(* IEC 61131-3 sources: SIMERLIFT/logiwork_simerlift_80v/logiwork_simerlift_80v/HEMAbattery/src_FBD/BCU, 8 files *)

(* ---- ampMaxTemp.iecst ---- *)
FUNCTION_BLOCK ampMultTemp {
    width := 200;
  }

VAR_INPUT
temp:REAL;
END_VAR

VAR_OUTPUT
mult : REAL;
END_VAR

VAR
rstTimer:TON;
timeout:BOOL;
lastMult:REAL;
instantMult:REAL;
END_VAR

IF temp<-20 THEN
	mult:=0;
	instantMult:=0;
ELSIF temp<-15  THEN
	instantMult:=0.1;
ELSIF temp<-10  THEN
	instantMult:=0.15;
ELSIF temp<-5  THEN
	instantMult:=0.2;
ELSIF temp<0  THEN
	instantMult:=0.4;
ELSIF temp<5  THEN
	instantMult:=0.5;
ELSIF temp<10  THEN
	instantMult:=0.7;
ELSIF temp<50  THEN
	instantMult:=1;
ELSIF temp<55  THEN
	instantMult:=0.4;
ELSIF temp<56  THEN
	instantMult:=0.2;
ELSE
	mult:=0;
	instantMult:=0;
END_IF;

rstTimer(IN:=instantMult=lastMult, PT:=T#10s, Q=>timeout);

lastMult:=instantMult;

IF timeout THEN
	mult:=instantMult;
END_IF;

END_FUNCTION_BLOCK

(* ---- ampMultVoltChar.iecst ---- *)
FUNCTION_BLOCK  ampMultVoltChar  {
    width := 200;
  }

VAR_INPUT
    chargeOn:BOOL;
    maxCell:UDINT;
END_VAR

VAR_OUTPUT
	mult:REAL;
END_VAR

VAR
state:USINT;

END_VAR

 IF NOT chargeOn THEN
    state:=0;
 END_IF;

 CASE state OF
	0:
	mult:=1;
	IF maxCell>3350 THEN
		state:=state+1;
	END_IF;

	1:
	mult:=0.7;
	IF maxCell>3400 THEN
		state:=state+1;
	END_IF;

	2:
	mult:=0.6;
	IF maxCell>3450 THEN
		state:=state+1;
	END_IF;

	3:
	mult:=0.5;
	IF maxCell>3500 THEN
		state:=state+1;
	END_IF;

	4:
	mult:=0.35;
	IF maxCell>3550 THEN
		state:=state+1;
	END_IF;

	5:
	mult:=0.3;
	IF maxCell>3600 THEN
		state:=state+1;
	END_IF;

	6:
	mult:=0.2;
	IF maxCell>3650 THEN
		state:=state+1;

	END_IF;

 	7:
	mult:=0;

END_CASE;

 END_FUNCTION_BLOCK

(* ---- ampMultVoltDisc.iecst ---- *)
FUNCTION_BLOCK  ampMultVoltDisc  {
    width := 200;
  }

VAR_INPUT
    discOn:BOOL;
    minCell:UDINT;
END_VAR

VAR_OUTPUT
	mult:REAL;
END_VAR

VAR
state:USINT;

END_VAR

 IF NOT discOn THEN
    state:=0;
 END_IF;

 CASE state OF
	0:
	mult:=1;
	IF minCell<3150 THEN
		state:=state+1;
	END_IF;

	1:
	mult:=0.7;
	IF minCell<3120 THEN
		state:=state+1;
	END_IF;

	2:
	mult:=0.6;
	IF minCell<3100 THEN
		state:=state+1;
	END_IF;

	3:
	mult:=0.5;
	IF minCell<3050 THEN
		state:=state+1;
	END_IF;

	4:
	mult:=0.35;
	IF minCell<3020 THEN
		state:=state+1;
	END_IF;

	5:
	mult:=0.25;
	IF minCell<3000 THEN
		state:=state+1;
	END_IF;

	6:
	mult:=0.2;
	IF minCell<2400 THEN
		state:=state+1;

	END_IF;

 	7:
	mult:=0;

END_CASE;

 END_FUNCTION_BLOCK

(* ---- bessState.iecst ---- *)
FUNCTION_BLOCK  bessState  {
    width := 400;
    bgColor := "mediumseagreen";
  }

VAR_INPUT
	IGNITION : BOOL;
	chargerON:BOOL;
	prechargeOk:BOOL;
	dischargeComplete:BOOL;
	chargeComplete:BOOL;
	shutdownComplete:BOOL;
	contactFbk:BOOL;
	currentAmp:REAL;
	OVfault:BOOL;
    UVfault:BOOL;
	fault:BOOL;
END_VAR

VAR_OUTPUT
	STATE : BATTSTATE;
	prechargeOn:BOOL;
	contact:BOOL;
	contactNeg:BOOL;
END_VAR

VAR
currentCharging:BOOL;
currentDischarging:BOOL;

CURRENTTIMERcharging:TON;
CURRENTTIMERdischarging:TON;

chargeVoltTimer:Tbuffer;
dischargeVoltTimer:Tbuffer;

BATTERYSTATE:BATTSTATE:=BATTSTATE#STANDBY;
PREVSTATE:BATTSTATE:=BATTSTATE#STANDBY;

BATTIMER:TON;
BATSTATEINTERVAL:TIME:=T#10s;
BATSTATETIMEOUT:BOOL;
BATSTATEELAPSEDTIME:TIME;
STANDBYINTERVAL:TIME:=T#2s;
END_VAR

CURRENTTIMERcharging(IN:=currentAmp<-0.5, PT:=T#500ms, Q=>currentCharging);
CURRENTTIMERdischarging(IN:=currentAmp>0.5, PT:=T#500ms, Q=>currentDischarging);
BATTIMER(IN:=BATTERYSTATE=PREVSTATE, PT:=BATSTATEINTERVAL, Q=>BATSTATETIMEOUT, ET=>BATSTATEELAPSEDTIME);

PREVSTATE:=BATTERYSTATE;

CASE BATTERYSTATE OF

	BATTSTATE#STANDBY:  // standby
		STATE:=BATTSTATE#STANDBY;
		BATSTATEINTERVAL:=T#12s;

		prechargeOn:=0;
		contact:=0;
		contactNeg:=0;

		// at the first time wait 2 sec
		IF BATSTATEELAPSEDTIME>STANDBYINTERVAL THEN
		    // then wait 100ms in next sessions
			STANDBYINTERVAL:=T#500ms;
			IF fault THEN
				BATTERYSTATE:=BATTSTATE#FAULT;
			ELSIF IGNITION THEN
				IF chargerON THEN
					IF OVfault OR chargeComplete THEN
						BATTERYSTATE:=BATTSTATE#CHARGECOMPLETE;
					ELSE
						BATTERYSTATE:=BATTSTATE#PRECHARGE;
					END_IF;
				ELSE
					BATTERYSTATE:=BATTSTATE#PRECHARGE;
				END_IF;
			END_IF;

		END_IF;

	BATTSTATE#PRECHARGE:  //discharge
		STATE:=BATTSTATE#PRECHARGE;
		BATSTATEINTERVAL:=T#5s;

		contactNeg:=1;

		IF BATSTATEELAPSEDTIME>T#50ms THEN
			prechargeOn:=1;
		ELSE
			prechargeOn:=0;
		END_IF;

		IF prechargeOk THEN
			contact:=1;
		ELSE
			contact:=0;
		END_IF;

		IF fault OR  NOT IGNITION  THEN
			BATTERYSTATE:=BATTSTATE#SHUTDOWN;
		ELSIF BATSTATETIMEOUT THEN
			BATTERYSTATE:=BATTSTATE#FAULT;
		ELSIF prechargeOk AND contactFbk THEN
			IF chargerON THEN
				IF OVfault OR chargeComplete THEN
					BATTERYSTATE:=BATTSTATE#CHARGECOMPLETE;
				ELSE
					BATTERYSTATE:=BATTSTATE#CHARGE;
				END_IF;
			ELSE
				BATTERYSTATE:=BATTSTATE#DISCHARGE;
			END_IF;
		END_IF;

	BATTSTATE#DISCHARGE:  //discharge
		STATE:=BATTSTATE#DISCHARGE;
		BATSTATEINTERVAL:=T#120s;

		prechargeOn:=0;
		contact:=1;
		contactNeg:=1;

		IF fault OR NOT IGNITION THEN
			BATTERYSTATE:=BATTSTATE#SHUTDOWN;
		ELSIF chargerON THEN
			IF OVfault OR chargeComplete THEN
				BATTERYSTATE:=BATTSTATE#CHARGECOMPLETE;
			ELSE
				BATTERYSTATE:=BATTSTATE#CHARGE;
			END_IF;
		ELSIF BATSTATEELAPSEDTIME>T#10s THEN
			IF currentDischarging THEN
				IF UVfault OR dischargeComplete THEN
					BATTERYSTATE:=BATTSTATE#DISCHARGECOMPLETE;
				END_IF;
			ELSIF currentCharging THEN
				IF OVfault THEN
					BATTERYSTATE:=BATTSTATE#CHARGECOMPLETE;
				END_IF;
			END_IF;
		ELSIF (UVfault OR dischargeComplete) AND currentAmp>10THEN
			BATTERYSTATE:=BATTSTATE#DISCHARGECOMPLETE;
		ELSIF (OVfault OR chargeComplete) AND currentAmp<-10 THEN
			BATTERYSTATE:=BATTSTATE#CHARGECOMPLETE;
		END_IF;

	BATTSTATE#CHARGE:  // charge
		STATE:=BATTSTATE#CHARGE;
		BATSTATEINTERVAL:=T#120s;

		prechargeOn:=0;
		contact:=1;
		contactNeg:=1;

		IF fault OR NOT IGNITION THEN
			BATTERYSTATE:=BATTSTATE#SHUTDOWN;
		ELSIF NOT chargerON THEN
			IF UVfault OR  dischargeComplete THEN
				BATTERYSTATE:=BATTSTATE#DISCHARGECOMPLETE;
			ELSE
				BATTERYSTATE:=BATTSTATE#DISCHARGE;
			END_IF;
		ELSIF OVfault OR chargeComplete THEN
			BATTERYSTATE:=BATTSTATE#CHARGECOMPLETE;
		ELSIF  BATSTATEELAPSEDTIME>T#8s THEN
			IF currentDischarging THEN
				IF UVfault THEN
					BATTERYSTATE:=BATTSTATE#DISCHARGECOMPLETE;
				ELSIF dischargeComplete THEN
					BATTERYSTATE:=BATTSTATE#DISCHARGECOMPLETE;
				END_IF;
			END_IF;
		ELSIF (UVfault OR dischargeComplete) AND currentAmp>10THEN
			BATTERYSTATE:=BATTSTATE#DISCHARGECOMPLETE;
		END_IF;

	BATTSTATE#SHUTDOWN:  // shutdown
		STATE:=BATTSTATE#SHUTDOWN;
		BATSTATEINTERVAL:=T#3000ms;
		prechargeOn:=0;
		IF BATSTATEELAPSEDTIME>T#2500ms OR  (shutdownComplete AND (BATSTATEELAPSEDTIME>T#1000ms))  THEN
			contact:=0;
		 	contactNeg:=0;
		 	IF contactFbk=FALSE THEN
				IF fault THEN
					BATTERYSTATE:=BATTSTATE#FAULT;
				ELSIF UVfault THEN
					BATTERYSTATE:=BATTSTATE#DISCHARGECOMPLETE;
				ELSIF OVfault THEN
					BATTERYSTATE:=BATTSTATE#CHARGECOMPLETE;
				ELSIF NOT IGNITION THEN
					BATTERYSTATE:=BATTSTATE#STANDBY;
				END_IF;
			ELSIF BATSTATEELAPSEDTIME>T#2800ms THEN
				BATTERYSTATE:=BATTSTATE#FAULT;
			END_IF;

		END_IF;

	BATTSTATE#FAULT:  //fault
		STATE:=BATTSTATE#FAULT;
		BATSTATEINTERVAL:=T#10s;

		prechargeOn:=0;
		contact:=0;
		contactNeg:=0;

		IF NOT fault AND (NOT IGNITION OR BATSTATETIMEOUT) THEN
			BATTERYSTATE:=BATTSTATE#STANDBY;
		END_IF;

	BATTSTATE#CHARGECOMPLETE:  //charge complete
		STATE:=BATTSTATE#CHARGECOMPLETE;
		BATSTATEINTERVAL:=T#5s;

		prechargeOn:=0;
		contact:=0;
		contactNeg:=0;

		IF fault OR NOT IGNITION THEN
			BATTERYSTATE:=BATTSTATE#SHUTDOWN;
		ELSIF NOT chargerON AND BATSTATETIMEOUT THEN
			IF UVfault THEN
				BATTERYSTATE:=BATTSTATE#DISCHARGECOMPLETE;
			ELSIF dischargeComplete THEN
				BATTERYSTATE:=BATTSTATE#DISCHARGECOMPLETE;
			ELSE
				BATTERYSTATE:=BATTSTATE#PRECHARGE;
			END_IF;
		END_IF;

	BATTSTATE#DISCHARGECOMPLETE:  //charge complete
		STATE:=BATTSTATE#DISCHARGECOMPLETE;
		BATSTATEINTERVAL:=T#5s;

		prechargeOn:=0;
		contact:=0;
		contactNeg:=0;

		IF fault THEN
			BATTERYSTATE:=BATTSTATE#SHUTDOWN;
		ELSIF NOT IGNITION THEN
			BATTERYSTATE:=BATTSTATE#SHUTDOWN;
		ELSIF chargerON AND BATSTATETIMEOUT THEN
			IF OVfault THEN
				BATTERYSTATE:=BATTSTATE#CHARGECOMPLETE;
			ELSIF chargeComplete THEN
				BATTERYSTATE:=BATTSTATE#CHARGECOMPLETE;
			ELSE
				BATTERYSTATE:=BATTSTATE#PRECHARGE;   /// because no current will flow unless contact closed
			END_IF;
		END_IF;

END_CASE;

END_FUNCTION_BLOCK

(* ---- chargeState.iecst ---- *)
FUNCTION_BLOCK  chargeState  {
    width := 400;
  }

VAR_INPUT
    chargeOn:BOOL;
    mainComplete:BOOL;
    dmcc:REAL;
	battAmpr:REAL;
	balAmpr:REAL;
	balDiff:UDINT;
    maxCell:UDINT;
    minCell:UDINT;
END_VAR

VAR_OUTPUT
	complete:BOOL;
	balance:BOOL;
	chargeAmpr:REAL;
	chState:USINT;
END_VAR

VAR

balDiffTol:UDINT;

balanceOK_mid:BOOL;
balanceOK:BOOL;
balanceTIMERhigh:TON;
balanceTIMERlow:TOF;

amperLow_mid:BOOL;
amperLow:BOOL;
amperTIMERhigh:TON;
amperTIMERlow:TOF;

PREVSTATE:USINT:=0;
state:USINT;
chargeTIMER:TON;
chargeInterval:TIME:=T#1s;
chargeSTATETIMEOUT:BOOL;
chargeSTATEELAPSEDTIME:TIME;
END_VAR

chargeTIMER(IN:=state=PREVSTATE, PT:=chargeInterval, Q=>chargeSTATETIMEOUT, ET=>chargeSTATEELAPSEDTIME);
PREVSTATE:=state;

amperTIMERhigh(IN:=ABS(battAmpr)<(balAmpr+3), PT:=T#3s, Q=>amperLow_mid);
amperTIMERlow(IN:=amperLow_mid, PT:=T#3s, Q=>amperLow);

balanceTIMERhigh(IN:= (maxCell-minCell)<balDiffTol, PT:=T#5s, Q=>balanceOK_mid);  //20
balanceTIMERlow(IN:=balanceOK_mid, PT:=T#5s, Q=>balanceOK);  //20

 IF NOT chargeOn THEN
    state:=0;
END_IF;

CASE state OF

	0: //stb
	chargeInterval:=T#5m;
	complete:=mainComplete;
	balance:=0;
	chargeAmpr:=dmcc;

	IF chargeOn AND NOT complete THEN
		state:=1;
		complete:=0;
	END_IF;

	1: //charge on
	chargeInterval:=T#5m;  //5m
	complete:=0;
	balance:=0;
	chargeAmpr:=dmcc;
	IF mainComplete THEN
		state:=2;  // go to rest before balance decision
	END_IF;

	2:  //rest
	chargeInterval:=T#10s;  //2m
	complete:=0;
	balance:=0;
	chargeAmpr:=balAmpr;
	balDiffTol:=balDiff;

	IF chargeSTATETIMEOUT THEN
		IF balanceOK THEN
			state:=4;
		ELSE
			state:=3;
		END_IF;
	ELSIF chargeSTATEELAPSEDTIME>T#30s THEN
		IF NOT amperLow THEN
			state:=4;
		END_IF;
	END_IF;

	3:  //balance
	chargeInterval:=T#1m;  //30m
	complete:=0;
	balance:=1;
	chargeAmpr:=balAmpr;
	balDiffTol:=10;

	IF chargeSTATETIMEOUT OR NOT amperLow THEN
		state:=4;
	ELSIF chargeSTATEELAPSEDTIME>T#10m THEN   //10m
		IF balanceOK THEN
			state:=4;
		END_IF;
	END_IF;

	4: //charge state complete
	chargeInterval:=T#1m;   //1m
	complete:=1;
	balance:=0;
	chargeAmpr:=0;

END_CASE;

chState:=state;

END_FUNCTION_BLOCK

(* ---- Current.iecfbd ---- *)
FUNCTION_BLOCK Current
  {
    Current {index := 0};
    Discharge_Current {index := 0};
    Charge_Current {index := 1};
    width := 300;
    height := 38;
  }

  VAR_INPUT
    Current : REAL := 0;
  END_VAR
  VAR_OUTPUT
    Charge_Current : UINT := 0;
    Discharge_Current : UINT := 0;
  END_VAR

  (*

    // Network 1:
    DIV(IN1 := Current, IN2 := 1000, DIV => @C(2).DIV);
    GE(IN1 := @C(2).DIV, IN2 := 0, GE => @C(11).GE);
    SEL_REAL(G := @C(11).GE, IN0 := 0, IN1 := @C(2).DIV, SEL_REAL => @C(19).SEL_REAL);
    TO_UINT(IN := @C(19).SEL_REAL, TO_UINT => Discharge_Current);
    LT(IN1 := @C(2).DIV, IN2 := 0, LT => @C(15).LT);
    MUL(IN1 := @C(2).DIV, IN2 := -1, MUL => @C(34).MUL);
    SEL_REAL(G := @C(15).LT, IN0 := 0, IN1 := @C(34).MUL, SEL_REAL => @C(27).SEL_REAL);
    TO_UINT(IN := @C(27).SEL_REAL, TO_UINT => Charge_Current);

  *)

  @VF(1) : @E(Current), @R(20.0, 20.0, 220.0, 19.0);
  @VF(4) : @E(Charge_Current), @R(1100.0, 80.0, 220.0, 19.0);
  @VF(5) : @E(Discharge_Current), @R(1100.0, 20.0, 220.0, 19.0);
  @C(11) : @F(GE), @R(550.0, 20.0, 40.0, 38.0), REAL, @I(@N(IN1), @L(9.5)), @I(@N(IN2), @L(29.5)), @O(@N(GE), @R(9.5));
  @VF(13) : @E(0), @R(360.0, 40.0, 110.0, 19.0), REAL;
  @C(15) : @F(LT), @R(550.0, 80.0, 40.0, 38.0), REAL, @I(@N(IN1), @L(9.5)), @I(@N(IN2), @L(29.5)), @O(@N(LT), @R(9.5));
  @VF(17) : @E(0), @R(360.0, 100.0, 110.0, 19.0), REAL;
  @C(19) : @F(SEL_REAL), @R(780.0, 20.0, 120.0, 58.0), @I(@N(G), @L(9.5)), @I(@N(IN0), @L(29.5)), @I(@N(IN1), @L(49.5)), @O(@N(SEL_REAL), @R(9.5));
  @VF(21) : @E(0), @R(630.0, 40.0, 110.0, 19.0), REAL;
  @C(24) : @F(TO_UINT), @R(940.0, 20.0, 120.0, 18.0), REAL, @I(@N(IN), @L(9.5)), @O(@N(TO_UINT), @R(9.5));
  @C(27) : @F(SEL_REAL), @R(780.0, 80.0, 120.0, 58.0), @I(@N(G), @L(9.5)), @I(@N(IN0), @L(29.5)), @I(@N(IN1), @L(49.5)), @O(@N(SEL_REAL), @R(9.5));
  @VF(28) : @E(0), @R(630.0, 100.0, 110.0, 19.0), REAL;
  @C(31) : @F(TO_UINT), @R(940.0, 80.0, 120.0, 18.0), REAL, @I(@N(IN), @L(9.5)), @O(@N(TO_UINT), @R(9.5));
  @C(34) : @F(MUL), @R(550.0, 120.0, 40.0, 38.0), REAL, @I(@N(IN1), @L(9.5)), @I(@N(IN2), @L(29.5)), @O(@N(MUL), @R(9.5));
  @VF(37) : @E(-1), @R(360.0, 140.0, 110.0, 19.0), REAL;
  @C(2) : @F(DIV), @R(280.0, 20.0, 40.0, 38.0), REAL, @I(@N(IN1), @L(9.5)), @I(@N(IN2), @L(29.5)), @O(@N(DIV), @R(9.5));
  @VF(7) : @E(1000), @R(130.0, 40.0, 110.0, 19.0), REAL;
  @CP(16) : 509.5, 29.5;
  @CP(23) : 509.5, 69.5;
  @CP(35) : 509.5, 89.5;

  @G(6) :
     @L(@CP(16), @C(11).IN1),
     @L(@CP(16), @CP(23)),
     @L(@CP(23), @CP(35)),
     @L(@CP(23), @C(19).IN1),
     @L(@CP(35), @C(15).IN1),
     @L(@CP(35), @C(34).IN1),
     @L(@C(2).DIV, @CP(16))
    ;
  @G(14) :
     @L(@VF(13).o, @C(11).IN2)
    ;
  @G(18) :
     @L(@VF(17).o, @C(15).IN2)
    ;
  @G(20) :
     @L(@C(11).GE, @C(19).G)
    ;
  @G(22) :
     @L(@VF(21).o, @C(19).IN0)
    ;
  @G(25) :
     @L(@C(19).SEL_REAL, @C(24).IN)
    ;
  @G(26) :
     @L(@C(24).TO_UINT, @VF(5).i)
    ;
  @G(29) :
     @L(@VF(28).o, @C(27).IN0)
    ;
  @G(30) :
     @L(@C(15).LT, @C(27).G)
    ;
  @G(32) :
     @L(@C(27).SEL_REAL, @C(31).IN)
    ;
  @G(33) :
     @L(@C(31).TO_UINT, @VF(4).i)
    ;
  @G(36) :
     @L(@C(34).MUL, @C(27).IN1)
    ;
  @G(38) :
     @L(@VF(37).o, @C(34).IN2)
    ;
  @G(3) :
     @L(@VF(1).o, @C(2).IN1)
    ;
  @G(8) :
     @L(@VF(7).o, @C(2).IN2)
    ;
END_FUNCTION_BLOCK

(* ---- essState1.iecst ---- *)
FUNCTION_BLOCK  essState1  {
    fault {index := 12};
    shutdownComplete {index := 11};
    chargeProtect {index := 9};
    dischargeProtect {index := 8};
    contactFbkNeg {loc := "left", index := 6};
    contactFbk {loc := "left", index := 5};
    prechargeOk {loc := "left", index := 4};
    contactNeg {loc := "right", index := 4};
    contact {loc := "right", index := 3};
    prechargeOn {loc := "right", index := 2};
    width := 400;
    bgColor := "mediumseagreen";
    height := 258;
  }

VAR_INPUT
	discharge:BOOL;
	charge:BOOL;
	shutdown:BOOL;

	prechargeOk:BOOL;
	contactFbk:BOOL;
	contactFbkNeg:BOOL;

	dischargeProtect:BOOL;
	chargeProtect:BOOL;

	shutdownComplete:BOOL;
	fault:BOOL;
END_VAR

VAR_OUTPUT
	STATE : BATTSTATE;

	prechargeOn:BOOL;
	contact:BOOL;
	contactNeg:BOOL;
END_VAR

VAR

BATTERYSTATE:BATTSTATE:=BATTSTATE#STANDBY;
PREVSTATE:BATTSTATE:=BATTSTATE#STANDBY;

BATTIMER:TON;
BATSTATEINTERVAL:TIME:=T#10s;
BATSTATETIMEOUT:BOOL;
BATSTATEELAPSEDTIME:TIME;
STANDBYINTERVAL:TIME:=T#2s;
END_VAR

BATTIMER(IN:=BATTERYSTATE=PREVSTATE, PT:=BATSTATEINTERVAL, Q=>BATSTATETIMEOUT, ET=>BATSTATEELAPSEDTIME);

PREVSTATE:=BATTERYSTATE;

CASE BATTERYSTATE OF

	BATTSTATE#STANDBY:  // standby
		STATE:=BATTSTATE#STANDBY;
		BATSTATEINTERVAL:=T#12s;

		contact:=0;
		contactNeg:=0;
		prechargeOn:=0;

        IF BATSTATEELAPSEDTIME>STANDBYINTERVAL THEN
        	STANDBYINTERVAL:=T#500ms;
        	IF fault THEN
				BATTERYSTATE:=BATTSTATE#FAULT;
			ELSIF shutdown THEN
				BATTERYSTATE:=BATTSTATE#SHUTDOWN;
			ELSIF discharge OR (charge AND NOT chargeProtect) THEN
				BATTERYSTATE:=BATTSTATE#PRECHARGE;
			END_IF;
        END_IF;

	BATTSTATE#PRECHARGE:  //discharge
		STATE:=BATTSTATE#PRECHARGE;
		BATSTATEINTERVAL:=T#5s;

		contactNeg:=1;

		IF BATSTATEELAPSEDTIME>T#50ms AND contactFbkNeg THEN
			prechargeOn:=1;
		END_IF;

		IF prechargeOk THEN
			contact:=1;
		END_IF;

		IF fault OR NOT(discharge OR charge) OR shutdown OR BATSTATETIMEOUT THEN
			BATTERYSTATE:=BATTSTATE#SHUTDOWN;
		ELSIF prechargeOk AND contactFbk AND contactFbkNeg THEN
			IF charge THEN
				BATTERYSTATE:=BATTSTATE#CHARGE;
			ELSE
				BATTERYSTATE:=BATTSTATE#DISCHARGE;
			END_IF;
		END_IF;

	BATTSTATE#DISCHARGE:  //discharge
		STATE:=BATTSTATE#DISCHARGE;
		BATSTATEINTERVAL:=T#120s;

		prechargeOn:=0;
		contact:=1;
		contactNeg:=1;

		IF fault OR shutdown OR NOT contactFbk OR NOT contactFbkNeg THEN
			BATTERYSTATE:=BATTSTATE#SHUTDOWN;
		ELSIF NOT discharge THEN
			IF charge AND NOT chargeProtect THEN
				BATTERYSTATE:=BATTSTATE#CHARGE;
			ELSE
				BATTERYSTATE:=BATTSTATE#SHUTDOWN;
			END_IF;
		END_IF;

	BATTSTATE#CHARGE:  // charge
		STATE:=BATTSTATE#CHARGE;
		BATSTATEINTERVAL:=T#120s;

		prechargeOn:=0;
		contact:=1;
		contactNeg:=1;

		IF fault OR shutdown OR NOT contactFbk OR NOT contactFbkNeg THEN
			BATTERYSTATE:=BATTSTATE#SHUTDOWN;
		ELSIF NOT charge THEN
			IF discharge THEN
				BATTERYSTATE:=BATTSTATE#DISCHARGE;
			ELSE
				BATTERYSTATE:=BATTSTATE#SHUTDOWN;
			END_IF;
		END_IF;

	BATTSTATE#SHUTDOWN:  // shutdown
		STATE:=BATTSTATE#SHUTDOWN;
		BATSTATEINTERVAL:=T#5000ms;

		prechargeOn:=0;

		IF shutdown OR BATSTATEELAPSEDTIME>T#2000ms OR (shutdownComplete AND (BATSTATEELAPSEDTIME>T#500ms))  THEN
			contact:=0;
			contactNeg:=0;
			IF fault THEN
				BATTERYSTATE:=BATTSTATE#FAULT;
			ELSIF shutdown THEN
				BATTERYSTATE:=BATTSTATE#SHUTDOWN;
			ELSIF NOT contactFbk AND NOT contactFbkNeg THEN
				IF dischargeProtect THEN
					BATTERYSTATE:=BATTSTATE#DISCHARGECOMPLETE;
				ELSIF chargeProtect THEN
					BATTERYSTATE:=BATTSTATE#CHARGECOMPLETE;
				ELSIF BATSTATETIMEOUT OR charge OR discharge THEN
					BATTERYSTATE:=BATTSTATE#STANDBY;
				END_IF;
			END_IF;
		END_IF;

	BATTSTATE#FAULT:  //fault
		STATE:=BATTSTATE#FAULT;
		BATSTATEINTERVAL:=T#10s;

		contact:=0;
		contactNeg:=0;
		prechargeOn:=0;

		IF NOT fault AND BATSTATETIMEOUT THEN
			BATTERYSTATE:=BATTSTATE#SHUTDOWN;
		END_IF;

	BATTSTATE#CHARGECOMPLETE:
		STATE:=BATTSTATE#CHARGECOMPLETE;
		BATSTATEINTERVAL:=T#5s;

		prechargeOn:=0;
		contact:=0;
		contactNeg:=0;

		IF fault THEN
			BATTERYSTATE:=BATTSTATE#FAULT;
		ELSIF shutdown THEN
			BATTERYSTATE:=BATTSTATE#SHUTDOWN;
		ELSIF BATSTATETIMEOUT AND discharge THEN
			BATTERYSTATE:=BATTSTATE#STANDBY;
		END_IF;

	BATTSTATE#DISCHARGECOMPLETE:
		STATE:=BATTSTATE#DISCHARGECOMPLETE;
		BATSTATEINTERVAL:=T#5s;

		prechargeOn:=0;
		contact:=0;
		contactNeg:=0;

		IF fault THEN
			BATTERYSTATE:=BATTSTATE#FAULT;
		ELSIF shutdown THEN
			BATTERYSTATE:=BATTSTATE#SHUTDOWN;
		ELSIF BATSTATETIMEOUT AND charge THEN
			BATTERYSTATE:=BATTSTATE#STANDBY;
		END_IF;

END_CASE;

END_FUNCTION_BLOCK

(* ---- GUI.iecfbd ---- *)
FUNCTION_BLOCK GUI
  {
    SoC {index := 0};
    SoH {index := 1};
    Voltage {index := 2};
    Current {index := 3};
    Temp {index := 4};
    Humidity {index := 5};
    Fault {index := 6};
    width := 200;
    height := 138;
  }

  VAR
    TP1 : TP;
    BAMTX2 : BAMTX;
    BATTSTACKinfo1 : BATTSTACKinfo;
    CANRECV5 : CANRECV;
    tauxCells : ARRAY[0..15] OF USINT := [0,0,0,1,1,1,2,2,2,3,3,3,4,4,4,4];
    guiReqCount : UDINT;
  END_VAR
  VAR_INPUT
    Voltage : REAL := 0;
    Current : REAL := 0;
    Temp : REAL := 0;
    Humidity : REAL := 0;
    Fault : UDINT := 0;
    SoC : USINT := 0;
    SoH : USINT := 0;
    Cycle : UINT;
    State : USINT;
    ID : USINT;
    CH : TMS570_CAN;
  END_VAR

  (*

    // Network 1:
    CANRECV5(CH := CH, ID := 16#18EA1EA4, FMT := CAN_FORMAT#EXTENDED, PER := T#1s, ENB := 1);
    RBIT(start := 0, len := 16, INbit := CANRECV5.DATA, OUTbit => @C(31).OUTbit);
    TO_UINT(IN := @C(31).OUTbit, TO_UINT => @C(2560).TO_UINT);
    FROM_BIG_ENDIAN(IN := @C(2560).TO_UINT, FROM_BIG_ENDIAN => @C(774).FROM_BIG_ENDIAN);
    RBIT(start := 8, len := 8, INbit := CANRECV5.DATA, OUTbit => @C(35).OUTbit);
    TO_USINT(IN := @C(35).OUTbit, TO_USINT => @C(2558).TO_USINT);
    RBIT(start := 0, len := 4, INbit := CANRECV5.DATA, OUTbit => @C(36).OUTbit);
    TO_USINT(IN := @C(36).OUTbit, TO_USINT => @C(2559).TO_USINT);
    DIV(IN1 := Voltage, IN2 := 1000, DIV => @C(988).DIV);
    DIV(IN1 := Current, IN2 := 1000, DIV => @C(12).DIV);
    TO_SINT(IN := Temp, TO_SINT => @C(799).TO_SINT);
    TO_USINT(IN := Humidity, TO_USINT => @C(820).TO_USINT);
    RBIT(start := 4, len := 4, INbit := CANRECV5.DATA, OUTbit => @C(29).OUTbit);
    TO_USINT(IN := @C(29).OUTbit, TO_USINT => @C(27).TO_USINT);
    EQ(IN1 := @C(27).TO_USINT, IN2 := ID, EQ => @C(789).EQ);
    NE(IN1 := guiReqCount, IN2 := CANRECV5.CRX, NE => @C(2565).NE);
    SEL(G := @C(2565).NE, IN0 := guiReqCount, IN1 := CANRECV5.CRX, SEL => guiReqCount);
    AND(IN1 := @C(2565).NE, IN2 := @C(789).EQ, AND => @C(779).AND);
    BATTSTACKinfo1(INFO := @C(2558).TO_USINT, BRD := @C(2559).TO_USINT, volt := @C(988).DIV, amp := @C(12).DIV, Cycle := Cycle, State := State, SOC := SoC, SOH := SoH, temp := @C(799).TO_SINT, hum := @C(820).TO_USINT, fault := Fault, NTCBETA := 3950, NTCNOMT_KLV := 298.15, NTCNOMR_OHM := 10000.0, T_CELLS := tAuxCells, R := @C(779).AND);
    BAMTX2(CH := CH, TPCM := 16#18FFABCD, TPDT := 16#18FFABCE, PGN := @C(774).FROM_BIG_ENDIAN, FRMPER := T#50ms, DATA := BATTSTACKinfo1.DATA, LEN := BATTSTACKinfo1.LEN, R := BATTSTACKinfo1.R_OUT);
    TP1(IN := BAMTX2.R_END, PT := T#100ms);

  *)

  @C(771) : @FB(TP1), @R(1640.0, 100.0, 100.0, 38.0), @I(@N(IN), @L(9.5)), @I(@N(PT), @L(29.5)), @O(@N(Q), @R(9.5)), @O(@N(ET), @R(29.5));
  @C(2566) : @FB(BAMTX2), @R(1290.0, 60.0, 220.0, 158.0), @I(@N(CH), @L(9.5)), @I(@N(TPCM), @L(29.5)), @I(@N(TPDT), @L(49.5)), @I(@N(PGN), @L(69.5)), @I(@N(FRMPER), @L(89.5)), @I(@N(DATA), @L(109.5)), @I(@N(LEN), @L(129.5)), @I(@N(R), @L(149.5)), @O(@N(CTX), @R(9.5)), @O(@N(RC), @R(29.5)), @O(@N(R_END), @R(49.5));
  @C(774) : @F(FROM_BIG_ENDIAN), @R(1110.0, 120.0, 160.0, 18.0), UINT, @I(@N(IN), @L(9.5)), @O(@N(FROM_BIG_ENDIAN), @R(9.5));
  @C(779) : @F(AND), @R(910.0, 460.0, 40.0, 38.0), BOOL, @I(@N(IN1), @L(9.5)), @I(@N(IN2), @L(29.5)), @O(@N(AND), @R(9.5));
  @C(789) : @F(EQ), @R(850.0, 480.0, 40.0, 38.0), USINT, @I(@N(IN1), @L(9.5)), @I(@N(IN2), @L(29.5)), @O(@N(EQ), @R(9.5));
  @C(799) : @F(TO_SINT), @R(840.0, 320.0, 110.0, 18.0), REAL, @I(@N(IN), @L(9.5)), @O(@N(TO_SINT), @R(9.5));
  @C(820) : @F(TO_USINT), @R(840.0, 340.0, 110.0, 18.0), REAL, @I(@N(IN), @L(9.5)), @O(@N(TO_USINT), @R(9.5));
  @C(2564) : @F(SEL), @R(690.0, 40.0, 120.0, 58.0), UDINT, @I(@N(G), @L(9.5)), @I(@N(IN0), @L(29.5)), @I(@N(IN1), @L(49.5)), @O(@N(SEL), @R(9.5));
  @C(2558) : @F(TO_USINT), @R(840.0, 160.0, 110.0, 18.0), LWORD, @I(@N(IN), @L(9.5)), @O(@N(TO_USINT), @R(9.5));
  @C(2559) : @F(TO_USINT), @R(840.0, 180.0, 110.0, 18.0), LWORD, @I(@N(IN), @L(9.5)), @O(@N(TO_USINT), @R(9.5));
  @C(2560) : @F(TO_UINT), @R(840.0, 120.0, 110.0, 18.0), LWORD, @I(@N(IN), @L(9.5)), @O(@N(TO_UINT), @R(9.5));
  @C(2565) : @F(NE), @R(410.0, 40.0, 40.0, 38.0), UDINT, @I(@N(IN1), @L(9.5)), @I(@N(IN2), @L(29.5)), @O(@N(NE), @R(9.5));
  @C(2567) : @FB(CANRECV5), @R(210.0, 120.0, 160.0, 98.0), @I(@N(CH), @L(9.5)), @I(@N(ID), @L(29.5)), @I(@N(FMT), @L(49.5)), @I(@N(PER), @L(69.5)), @I(@N(ENB), @L(89.5)), @O(@N(CRX), @R(9.5)), @O(@N(DATA), @R(29.5)), @O(@N(DLC), @R(49.5)), @O(@N(MPER), @R(69.5)), @O(@N(RC), @R(89.5));
  @VF(791) : @E(T#100ms), @R(1530.0, 120.0, 90.0, 19.0);
  @VF(2577) : @E(T#50ms), @R(1160.0, 140.0, 110.0, 19.0);
  @VF(2580) : @E(16#18FFABCE), @R(1050.0, 100.0, 220.0, 19.0), UDINT;
  @VF(2586) : @E(16#18FFABCD), @R(1050.0, 80.0, 220.0, 19.0), UDINT;
  @VF(2572) : @E(tAuxCells), @R(840.0, 440.0, 110.0, 19.0);
  @VF(2573) : @E(298.15), @R(840.0, 400.0, 110.0, 19.0), REAL;
  @VF(2575) : @E(10000.0), @R(840.0, 420.0, 110.0, 19.0), REAL;
  @VF(793) : @E(3950), @R(840.0, 380.0, 110.0, 19.0), REAL;
  @VF(837) : @E(guiReqCount), @R(480.0, 60.0, 110.0, 19.0);
  @VF(2581) : @E(0), @R(410.0, 100.0, 40.0, 19.0), INT;
  @VF(2583) : @E(8), @R(410.0, 180.0, 40.0, 19.0), INT;
  @VF(2582) : @E(8), @R(410.0, 160.0, 40.0, 19.0), INT;
  @VF(2578) : @E(16), @R(410.0, 120.0, 40.0, 19.0), INT;
  @VF(2585) : @E(4), @R(410.0, 240.0, 40.0, 19.0), INT;
  @VF(2584) : @E(0), @R(410.0, 220.0, 40.0, 19.0), INT;
  @VF(801) : @E(4), @R(410.0, 480.0, 40.0, 19.0), INT;
  @VF(802) : @E(4), @R(410.0, 500.0, 40.0, 19.0), INT;
  @VF(798) : @E(guiReqCount), @R(280.0, 40.0, 110.0, 19.0);
  @VF(2592) : @E(1), @R(80.0, 200.0, 110.0, 19.0), BOOL;
  @VF(2591) : @E(T#1s), @R(80.0, 180.0, 110.0, 19.0);
  @VF(2593) : @E(CAN_FORMAT#EXTENDED), @R(20.0, 160.0, 170.0, 19.0);
  @VF(2589) : @E(16#18EA1EA4), @R(20.0, 140.0, 170.0, 19.0), UDINT;
  @VF(1) : @E(Fault), @R(840.0, 360.0, 110.0, 19.0);
  @VF(2) : @E(Humidity), @R(730.0, 340.0, 90.0, 19.0);
  @VF(3) : @E(Temp), @R(730.0, 320.0, 90.0, 19.0);
  @VF(4) : @E(Current), @R(20.0, 320.0, 220.0, 19.0);
  @VF(5) : @E(Voltage), @R(20.0, 280.0, 220.0, 19.0);
  @VF(6) : @E(SoC), @R(840.0, 280.0, 110.0, 19.0);
  @VF(7) : @E(SoH), @R(840.0, 300.0, 110.0, 19.0);
  @C(988) : @F(DIV), @R(280.0, 280.0, 40.0, 38.0), REAL, @I(@N(IN1), @L(9.5)), @I(@N(IN2), @L(29.5)), @O(@N(DIV), @R(9.5));
  @VF(981) : @E(1000), @R(130.0, 300.0, 110.0, 19.0), REAL;
  @C(12) : @F(DIV), @R(280.0, 320.0, 40.0, 38.0), REAL, @I(@N(IN1), @L(9.5)), @I(@N(IN2), @L(29.5)), @O(@N(DIV), @R(9.5));
  @VF(16) : @E(1000), @R(130.0, 340.0, 110.0, 19.0), REAL;
  @VF(21) : @E(Cycle), @R(840.0, 240.0, 110.0, 19.0);
  @VF(22) : @E(State), @R(840.0, 260.0, 110.0, 19.0);
  @C(773) : @FB(BATTSTACKinfo1), @R(970.0, 160.0, 300.0, 318.0), @I(@N(INFO), @L(9.5)), @I(@N(BRD), @L(29.5)), @I(@N(volt), @L(49.5)), @I(@N(amp), @L(69.5)), @I(@N(Cycle), @L(89.5)), @I(@N(State), @L(109.5)), @I(@N(SOC), @L(129.5)), @I(@N(SOH), @L(149.5)), @I(@N(temp), @L(169.5)), @I(@N(hum), @L(189.5)), @I(@N(fault), @L(209.5)), @I(@N(NTCBETA), @L(229.5)), @I(@N(NTCNOMT_KLV), @L(249.5)), @I(@N(NTCNOMR_OHM), @L(269.5)), @I(@N(T_CELLS), @L(289.5)), @I(@N(R), @L(309.5)), @O(@N(DATA), @R(9.5)), @O(@N(LEN), @R(29.5)), @O(@N(R_OUT), @R(49.5));
  @VF(25) : @E(ID), @R(660.0, 500.0, 140.0, 19.0);
  @C(27) : @F(TO_USINT), @R(670.0, 480.0, 120.0, 18.0), LWORD, @I(@N(IN), @L(9.5)), @O(@N(TO_USINT), @R(9.5));
  @VF(32) : @E(CH), @R(10.0, 10.0, 140.0, 19.0);
  @C(31) : @F(RBIT), @R(470.0, 100.0, 120.0, 58.0), @I(@N(start), @L(9.5)), @I(@N(len), @L(29.5)), @I(@N(INbit), @L(49.5)), @O(@N(OUTbit), @R(9.5));
  @C(35) : @F(RBIT), @R(470.0, 160.0, 120.0, 58.0), @I(@N(start), @L(9.5)), @I(@N(len), @L(29.5)), @I(@N(INbit), @L(49.5)), @O(@N(OUTbit), @R(9.5));
  @C(36) : @F(RBIT), @R(470.0, 220.0, 120.0, 58.0), @I(@N(start), @L(9.5)), @I(@N(len), @L(29.5)), @I(@N(INbit), @L(49.5)), @O(@N(OUTbit), @R(9.5));
  @C(29) : @F(RBIT), @R(470.0, 480.0, 120.0, 58.0), @I(@N(start), @L(9.5)), @I(@N(len), @L(29.5)), @I(@N(INbit), @L(49.5)), @O(@N(OUTbit), @R(9.5));
  @CP(804) : 619.5, 49.5;
  @CP(2595) : 389.5, 149.5;
  @CP(58) : 389.5, 209.5;
  @CP(282) : 389.5, 269.5;
  @CP(333) : 389.5, 89.5;
  @CP(34) : 189.5, 19.5;

  @G(805) :
     @L(@VF(791).o, @C(771).PT)
    ;
  @G(825) :
     @L(@C(2566).R_END, @C(771).IN)
    ;
  @G(2612) :
     @L(@VF(2577).o, @C(2566).FRMPER)
    ;
  @G(2622) :
     @L(@VF(2580).o, @C(2566).TPDT)
    ;
  @G(2629) :
     @L(@VF(2586).o, @C(2566).TPCM)
    ;
  @G(828) :
     @L(@C(774).FROM_BIG_ENDIAN, @C(2566).PGN)
    ;
  @G(823) :
     @L(@C(773).DATA, @C(2566).DATA)
    ;
  @G(821) :
     @L(@C(773).LEN, @C(2566).LEN)
    ;
  @G(817) :
     @L(@C(773).R_OUT, @C(2566).R)
    ;
  @G(807) :
     @L(@C(799).TO_SINT, @C(773).temp)
    ;
  @G(834) :
     @L(@C(820).TO_USINT, @C(773).hum)
    ;
  @G(813) :
     @L(@VF(793).o, @C(773).NTCBETA)
    ;
  @G(814) :
     @L(@VF(2573).o, @C(773).NTCNOMT_KLV)
    ;
  @G(815) :
     @L(@VF(2575).o, @C(773).NTCNOMR_OHM)
    ;
  @G(816) :
     @L(@VF(2572).o, @C(773).T_CELLS)
    ;
  @G(824) :
     @L(@C(779).AND, @C(773).R)
    ;
  @G(819) :
     @L(@C(2559).TO_USINT, @C(773).BRD)
    ;
  @G(822) :
     @L(@C(2558).TO_USINT, @C(773).INFO)
    ;
  @G(829) :
     @L(@C(2560).TO_UINT, @C(774).IN)
    ;
  @G(2628) :
     @L(@C(2565).NE, @CP(804)),
     @L(@CP(804), @C(2564).G),
     @L(@CP(804), @C(779).IN1)
    ;
  @G(838) :
     @L(@VF(837).o, @C(2564).IN0)
    ;
  @G(2618) :
     @L(@C(2567).CRX, @CP(333)),
     @L(@CP(333), @C(2565).IN2),
     @L(@CP(333), @C(2564).IN1)
    ;
  @G(2621) :
     @L(@C(2567).DATA, @CP(2595)),
     @L(@CP(2595), @CP(58)),
     @L(@CP(58), @CP(282)),
     @L(@CP(282), @C(36).INbit),
     @L(@CP(58), @C(35).INbit),
     @L(@CP(2595), @C(31).INbit),
     @L(@CP(282), @C(29).INbit)
    ;
  @G(812) :
     @L(@VF(798).o, @C(2565).IN1)
    ;
  @G(836) :
     @L(@C(2564).SEL, @VF(798).i)
    ;
  @G(2633) :
     @L(@VF(2593).o, @C(2567).FMT)
    ;
  @G(2634) :
     @L(@VF(2589).o, @C(2567).ID)
    ;
  @G(2635) :
     @L(@VF(2591).o, @C(2567).PER)
    ;
  @G(2636) :
     @L(@VF(2592).o, @C(2567).ENB)
    ;
  @G(8) :
     @L(@VF(1).o, @C(773).fault)
    ;
  @G(9) :
     @L(@VF(3).o, @C(799).IN)
    ;
  @G(10) :
     @L(@VF(2).o, @C(820).IN)
    ;
  @G(13) :
     @L(@VF(6).o, @C(773).SOC)
    ;
  @G(14) :
     @L(@VF(7).o, @C(773).SOH)
    ;
  @G(15) :
     @L(@VF(981).o, @C(988).IN2)
    ;
  @G(11) :
     @L(@C(988).DIV, @C(773).volt)
    ;
  @G(17) :
     @L(@VF(16).o, @C(12).IN2)
    ;
  @G(18) :
     @L(@C(12).DIV, @C(773).amp)
    ;
  @G(19) :
     @L(@VF(4).o, @C(12).IN1)
    ;
  @G(20) :
     @L(@VF(5).o, @C(988).IN1)
    ;
  @G(23) :
     @L(@VF(21).o, @C(773).Cycle)
    ;
  @G(24) :
     @L(@VF(22).o, @C(773).State)
    ;
  @G(26) :
     @L(@VF(25).o, @C(789).IN2)
    ;
  @G(28) :
     @L(@C(27).TO_USINT, @C(789).IN1)
    ;
  @G(33) :
     @L(@VF(32).o, @CP(34)),
     @L(@CP(34), @C(2566).CH),
     @L(@CP(34), @C(2567).CH)
    ;
  @G(30) :
     @L(@C(789).EQ, @C(779).IN2)
    ;
  @G(37) :
     @L(@VF(2584).o, @C(36).start)
    ;
  @G(38) :
     @L(@VF(2585).o, @C(36).len)
    ;
  @G(39) :
     @L(@VF(2578).o, @C(31).len)
    ;
  @G(40) :
     @L(@VF(2581).o, @C(31).start)
    ;
  @G(41) :
     @L(@VF(2582).o, @C(35).start)
    ;
  @G(42) :
     @L(@VF(2583).o, @C(35).len)
    ;
  @G(43) :
     @L(@C(31).OUTbit, @C(2560).IN)
    ;
  @G(44) :
     @L(@C(35).OUTbit, @C(2558).IN)
    ;
  @G(45) :
     @L(@C(36).OUTbit, @C(2559).IN)
    ;
  @G(46) :
     @L(@VF(801).o, @C(29).start)
    ;
  @G(47) :
     @L(@VF(802).o, @C(29).len)
    ;
  @G(48) :
     @L(@C(29).OUTbit, @C(27).IN)
    ;
END_FUNCTION_BLOCK
